SUBAPPLICATION Uebung_011a_AX (* Numeric Value Output und BUTTON_PRESS_REPEAT_DONE *)
  (* Standard: 61499-2; Description: Copyright (c) 2023 Meisterschulen am Ostbahnhof This program and the accompanying materials are made available under the terms of the Eclipse Public License 2.0 which is available at https://www.eclipse.org/legal/epl-2.0/ SPDX-License-Identifier: EPL-2.0 *)
  (* Version 1.0, 2023-10-23, Franz Höpfinger, Meisterschulen am Ostbahnhof, initial API and implementation and/or initial documentation *)
  PACKAGE Uebungen;
  IMPORT Uebungen::const::UT::DefaultPool::OutputNumber_N1;
  IMPORT logiBUS::io::DI::logiBUS_DI::Input_I1;
  IMPORT logiBUS::io::DI::logiBUS_DI_Events::BUTTON_PRESS_REPEAT_DONE;
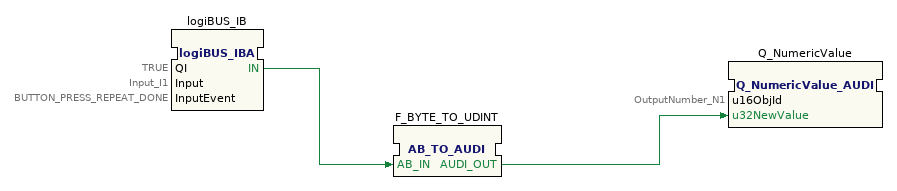
  (* BUTTON_PRESS_REPEAT_DONE: nur am Ende 1 Event BUTTON_PRESS_REPEAT: Während des drückens kommen Events *)
  FBS
    Q_NumericValue : isobus::UT::Q::Q_NumericValue_AUDI(u16ObjId := OutputNumber_N1);
    logiBUS_IB : logiBUS::io::DI::logiBUS_IBA(QI := TRUE, Input := Input_I1, InputEvent := BUTTON_PRESS_REPEAT_DONE);
    F_BYTE_TO_UDINT : adapter::conversion::unidirectional::AB_TO_AUDI;
  END_FBS
  ADAPTER_CONNECTIONS
    logiBUS_IB.IN TO F_BYTE_TO_UDINT.AB_IN;
    F_BYTE_TO_UDINT.AUDI_OUT TO Q_NumericValue.u32NewValue;
  END_CONNECTIONS
END_SUBAPPLICATION
